INTERFACE ITF_BaseLogger_HMI_Connector_View

(*			
	RafalOS
	Rafał Osajda		02.10.2025		TC 4024.66
	Zwraca czy nastąpiła jakaś zmiana w pamięci zgłoszeń - całej nie tylko dla jakiegoś elementu
*)
METHOD PUBLIC GetChangeInMemory : BOOL
VAR_INPUT
END_VAR
END_METHOD

METHOD PUBLIC GetEventCounts : ST_BaseEvents_ActiveEvents
VAR_INPUT
END_VAR
END_METHOD

METHOD PUBLIC GetEventCountsForItem : ST_BaseEvents_ActiveEvents
VAR_INPUT
	uiIDItem: UINT;
END_VAR
END_METHOD

METHOD PUBLIC GetInformationFromItem : ST_BaseLogger_ItemDataToDisplay
VAR_INPUT
	uiIDItem				: UINT;
	uiIDEvent				: UINT;
END_VAR
END_METHOD

METHOD GetReferenceToStmemory : REFERENCE TO ST_BaseEvents_Memory
VAR_INPUT
	
END_VAR
END_METHOD

(*			
	RafalOS
	Rafał Osajda		02.10.2025		TC 4024.66
	
*)
METHOD PUBLIC ResetChangeInMemory : BOOL
VAR_INPUT
END_VAR
END_METHOD

END_INTERFACE

(* stored: Version 1.1.0.1
   Itf ITF_BaseLogger_HMI_Connector_View: Id {77898fe0-1ee7-0a01-1a2c-9ed188780169}
   Method GetChangeInMemory: Id {cefe7588-5f63-083f-0636-0b6488cb4e6e}
   Method GetEventCounts: Id {515d209a-bf83-0d57-2f97-7f48446c4713}
   Method GetEventCountsForItem: Id {5a0b0f72-7e2e-0356-11bd-46b2df6bcce5}
   Method GetInformationFromItem: Id {e03af02b-30ef-08f3-2938-f43d70776345}
   Method GetReferenceToStmemory: Id {cd9afe9d-8904-045f-3d51-457b59128ac2}
   Method ResetChangeInMemory: Id {d381c273-43a8-0471-16dd-328c4ccf4ec4} *)
